(* IEC 61131-3 sources: Bob/Head_Pkg/ModuleControl, 4 files *)

(* ---- Types.typ ---- *)
TYPE
	PowerSupplyState_enum :
		(
		WAIT_FOR_READY_TO_POWER,
		WAIT_FOR_POWER_ON,
		READY,
		ERROR
		);
	localHead_typ : 	STRUCT
		pressureTransducerRaw : INT;
	END_STRUCT;
	localModule_typ : 	STRUCT
		ps : localPS_typ;
		valve : localValve_typ;
		supplyTemperatureRaw : INT;
		head : ARRAY[0..NUM_OF_HEADS_PER_MODULE_M1]OF localHead_typ;
	END_STRUCT;
	localPS_typ : 	STRUCT
		state : PowerSupplyState_enum;
		axis : ACP10AXIS_typ;
		mpAxis : UDINT;
		mpParams : MpAxisBasicParType;
		MpAxisBasic_0 : MpAxisBasic;
	END_STRUCT;
	localValve_typ : 	STRUCT
		valveName : STRING[80];
		outputModuleOk : BOOL; (*variable to be linked to the module ok on the IO module used for the outputs*)
		inputModuleOk : BOOL; (*variable to be linked to the module ok on the IO module used for the inputs*)
		doOpen : BOOL; (*variable to be linked to the digital output which opens the valve*)
		diOpened : BOOL; (*variable to be linked to the digital input which indicates that the valve is opened*)
		diClosed : BOOL; (*variable to be linked to the digital input which indicates that the valve is closed*)
		openDebounceTimer : TON;
		closeDebounceTimer : TON;
		openTime : REAL;
		openErrorTimer : TON;
		closeTime : REAL;
		closeErrorTimer : TON;
		MpRecipeRegPar_0 : MpRecipeRegPar;
		MpRecipeRegPar_1 : MpRecipeRegPar;
		openError_r_trig : r_trig;
		openError_f_trig : f_trig;
		closeError_r_trig : r_trig;
		closeError_f_trig : f_trig;
		open_and_close_error_r_trig : r_trig;
		open_and_close_error_f_trig : f_trig;
		io_error_r_trig : r_trig;
		io_error_f_trig : f_trig;
	END_STRUCT;
END_TYPE

(* ---- Main.st ---- *)
PROGRAM _INIT
    modules[0].valve.valveName := 'Module 1 Supply Valve';
    modules[1].valve.valveName := 'Module 2 Supply Valve';

    MpRecipeRegPar_0[0].PVName := ADR('gModules[0].heads[0].enable');
    MpRecipeRegPar_0[1].PVName := ADR('gModules[0].heads[1].enable');
    MpRecipeRegPar_0[2].PVName := ADR('gModules[1].heads[0].enable');
    MpRecipeRegPar_0[3].PVName := ADR('gModules[1].heads[1].enable');

    FOR currentHead:=0 TO NUMBER_OF_HEADS_M1 DO
        MpRecipeRegPar_0[currentHead].MpLink := ADR(gMachineRecipe);
        MpRecipeRegPar_0[currentHead].Enable := TRUE;
        MpRecipeRegPar_0[currentHead].Category := ADR(MACHINE_CATEGORY);
        MpRecipeRegPar_0[currentHead]();
    END_FOR

	gModules[0].productSupply.parameters;
    MpRecipeRegPar_1[0].PVName := ADR('gModules[0].productSupply.parameters');
    MpRecipeRegPar_1[1].PVName := ADR('gModules[1].productSupply.parameters');

    FOR currentHead:=0 TO NUMBER_OF_MODULES_M1 DO
        MpRecipeRegPar_1[currentHead].MpLink := ADR(gMachineRecipe);
        MpRecipeRegPar_1[currentHead].Enable := TRUE;
        MpRecipeRegPar_1[currentHead].Category := ADR(MACHINE_CATEGORY);
        MpRecipeRegPar_1[currentHead]();
    END_FOR

    MpRecipeRegPar_2[0].PVName := ADR('gModules[0].heads[0].pressureTransducer.parameters');
    MpRecipeRegPar_2[1].PVName := ADR('gModules[0].heads[1].pressureTransducer.parameters');
    MpRecipeRegPar_2[2].PVName := ADR('gModules[1].heads[0].pressureTransducer.parameters');
    MpRecipeRegPar_2[3].PVName := ADR('gModules[1].heads[1].pressureTransducer.parameters');

    FOR currentHead:=0 TO NUMBER_OF_HEADS_M1 DO
        MpRecipeRegPar_2[currentHead].MpLink := ADR(gMachineRecipe);
        MpRecipeRegPar_2[currentHead].Enable := TRUE;
        MpRecipeRegPar_2[currentHead].Category := ADR(MACHINE_CATEGORY);
        MpRecipeRegPar_2[currentHead]();
    END_FOR

END_PROGRAM

PROGRAM _CYCLIC

    memset(ADR(logArguments), 0, SIZEOF(logArguments));

	modules[0].ps.mpAxis := ADR(gMpAxisPS1);
	modules[1].ps.mpAxis := ADR(gMpAxisPS2);

	FOR currentModule:=0 TO NUMBER_OF_MODULES_M1 DO

        gModules[currentModule].productSupply.temperature   := ((modules[currentModule].supplyTemperatureRaw * gModules[currentModule].productSupply.parameters.scalingFactor) + gModules[currentModule].productSupply.parameters.scalingOffset) / 100.0;
        productSupplyValveAction;

        FOR currentHead:=0 TO NUM_OF_HEADS_PER_MODULE_M1 DO
			pCurrentHead ACCESS ADR(gModules[currentModule].heads[currentHead]);

			//set .ready bit for each head
            pCurrentHead.ready                          := ((pCurrentHead.stretchRod.status.atHome = TRUE OR pCurrentHead.stretchRod.status.atRetractPos= TRUE) AND (pCurrentHead.nozzle.status.opened = TRUE) AND ((pCurrentHead.fillPiston.status.atReturnPos = TRUE) OR (pCurrentHead.enable = FALSE)));
            pCurrentHead.pressureTransducer.pressure    := (modules[currentModule].head[currentHead].pressureTransducerRaw - pCurrentHead.pressureTransducer.parameters.scalingOffset) * pCurrentHead.pressureTransducer.parameters.scalingFactor;
        END_FOR

        logArguments[0] := ADR(currentModule);
        logArguments[1] := ADR(modules[currentModule].ps.MpAxisBasic_0.Info.HardwareInfo.NodeID);

        // if an error occurs in any state then go to the error state
        CASE modules[currentModule].ps.state OF
            ERROR:

            ELSE
                IF (modules[currentModule].ps.MpAxisBasic_0.Error = TRUE) THEN
                    logArguments[3] := ADR(modules[currentModule].ps.MpAxisBasic_0.StatusID);
                    logError('Power Supply', 'Module %h, Node %h Error %d', ADR(logArguments));
                    modules[currentModule].ps.state := ERROR;
                ELSIF (gModules[currentModule].powerSupply.commands.errorAcknowledge = TRUE) THEN
                    gModules[currentModule].powerSupply.commands.errorAcknowledge := FALSE;
                END_IF
        END_CASE

        CASE (modules[currentModule].ps.state) OF
            WAIT_FOR_READY_TO_POWER:
                IF (modules[currentModule].ps.MpAxisBasic_0.Info.AxisInitialized <> TRUE) AND (modules[currentModule].ps.MpAxisBasic_0.Update = FALSE) THEN
                    modules[currentModule].ps.MpAxisBasic_0.Update := TRUE;
                ELSIF (modules[currentModule].ps.MpAxisBasic_0.UpdateDone = TRUE) THEN
                    modules[currentModule].ps.MpAxisBasic_0.Update := FALSE;
                END_IF

                IF (modules[currentModule].ps.MpAxisBasic_0.Info.ReadyToPowerOn = TRUE) AND (gMachineControl.commands.powerOn = TRUE) THEN
					logArguments[0] := ADR(modules[currentModule].ps.MpAxisBasic_0.Info.HardwareInfo.NodeID);
					logDebug('PSControl', 'Power Supply Axis Ready to power on, index = %d', ADR(logArguments));
                    modules[currentModule].ps.MpAxisBasic_0.Power   := TRUE;
                    modules[currentModule].ps.state                 := WAIT_FOR_POWER_ON;
                END_IF

			WAIT_FOR_POWER_ON:
                IF (modules[currentModule].ps.MpAxisBasic_0.PowerOn = TRUE) THEN
                    logArguments[0] := ADR(modules[currentModule].ps.MpAxisBasic_0.Info.HardwareInfo.NodeID);
                    logDebug('PSControl', 'Node %d Power Supply Axis powered on', ADR(logArguments));
                    modules[currentModule].ps.state := READY;
                END_IF

            READY:
                IF (gMachineControl.commands.powerOn = FALSE) THEN
                    modules[currentModule].ps.MpAxisBasic_0.Power   := FALSE;
                    logArguments[0] := ADR(modules[currentModule].ps.MpAxisBasic_0.Info.HardwareInfo.NodeID);
                    logDebug('PSControl', 'Node %d Power Supply Axis powered off', ADR(logArguments));
                    modules[currentModule].ps.state := WAIT_FOR_READY_TO_POWER;
                END_IF

            ERROR:
                IF (gModules[currentModule].powerSupply.commands.errorAcknowledge = TRUE) THEN
                    logDebug('FillPiston', 'Module %h, Head %h, Node %h Acknowledging Error', ADR(logArguments));
                    gModules[currentModule].powerSupply.commands.errorAcknowledge   := FALSE;
                    modules[currentModule].ps.MpAxisBasic_0.ErrorReset                 := TRUE;
                END_IF

                IF (modules[currentModule].ps.MpAxisBasic_0.Error <> TRUE) THEN
                    logDebug('PSControl', 'Module %h, Node %h All Errors Acknowledged', ADR(logArguments));
                    modules[currentModule].ps.MpAxisBasic_0.ErrorReset  := FALSE;
                    IF (modules[currentModule].ps.MpAxisBasic_0.PowerOn = TRUE) THEN
                        modules[currentModule].ps.state := READY;
                    ELSE
                        modules[currentModule].ps.state := WAIT_FOR_READY_TO_POWER;
                    END_IF
                END_IF
        END_CASE

        IF (modules[currentModule].ps.state <> old_state[currentModule]) THEN
            old_state[currentModule] := modules[currentModule].ps.state;
            logArguments[0] := ADR(modules[currentModule].ps.MpAxisBasic_0.Info.HardwareInfo.NodeID);
            logArguments[1] := ADR(modules[currentModule].ps.state);
            logDebug('PSControl', 'Node %d Changing State to %d', ADR(logArguments));
        END_IF

        modules[currentModule].ps.MpAxisBasic_0.Enable      := TRUE;
        modules[currentModule].ps.MpAxisBasic_0.Axis        := ADR(modules[currentModule].ps.axis);
        modules[currentModule].ps.MpAxisBasic_0.MpLink      := modules[currentModule].ps.mpAxis;
        modules[currentModule].ps.MpAxisBasic_0.Parameters  := ADR(modules[currentModule].ps.mpParams);
        modules[currentModule].ps.MpAxisBasic_0();

        gModules[currentModule].powerSupply.status.errorActive  := modules[currentModule].ps.MpAxisBasic_0.Error;
        gModules[currentModule].powerSupply.status.errorNumber  := modules[currentModule].ps.MpAxisBasic_0.StatusID;
        gModules[currentModule].powerSupply.status.poweredOn    := modules[currentModule].ps.MpAxisBasic_0.PowerOn;

	END_FOR

END_PROGRAM

PROGRAM _EXIT
    FOR currentModule:=0 TO NUMBER_OF_MODULES_M1 DO
        modules[currentModule].ps.MpAxisBasic_0.Enable  := FALSE;
        modules[currentModule].ps.MpAxisBasic_0();
    END_FOR
END_PROGRAM

(* ---- productSupplyVavle.st ---- *)
ACTION productSupplyValveAction:

    pCurrentValve ACCESS ADR(gModules[currentModule].productSupply.valve);
    pLocalValve ACCESS ADR(modules[currentModule].valve);

    IF (pCurrentValve.parameters.machineData.enabled = TRUE) THEN

        IF (((pCurrentValve.commands.open = TRUE) AND (pCurrentValve.commands.close = FALSE)) AND
            (pLocalValve.doOpen = FALSE)) THEN
            logDebug('Fill Valve', 'Module %h, Head %h, Open Command', ADR(logArguments));
            pLocalValve.doOpen := TRUE;
        END_IF

        IF (((pCurrentValve.commands.close = TRUE) AND (pCurrentValve.commands.open = FALSE)) AND
            (pLocalValve.doOpen = TRUE)) THEN
            logDebug('Fill Valve', 'Module %h, Head %h, Close Command', ADR(logArguments));
            pLocalValve.doOpen := FALSE;
        END_IF

        // 20ms debounce timer
        pLocalValve.openDebounceTimer.IN    := pLocalValve.diOpened;
        pLocalValve.openDebounceTimer.PT    := pCurrentValve.parameters.machineData.debounceTime;
        pLocalValve.openDebounceTimer();

        // 20ms debounce timer
        pLocalValve.closeDebounceTimer.IN := pLocalValve.diClosed;
        pLocalValve.closeDebounceTimer.PT := pCurrentValve.parameters.machineData.debounceTime;
        pLocalValve.closeDebounceTimer();

        // ensure that the valve opens
        pLocalValve.openErrorTimer.IN    := ((pCurrentValve.commands.open = TRUE) AND (pLocalValve.diOpened = FALSE));
        pLocalValve.openErrorTimer.PT    := pCurrentValve.parameters.machineData.timeout;
        pLocalValve.openErrorTimer();

        // ensure that the valve closes
        pLocalValve.closeErrorTimer.IN := ((pCurrentValve.commands.close = TRUE) AND (pLocalValve.diClosed = FALSE));
        pLocalValve.closeErrorTimer.PT := pCurrentValve.parameters.machineData.timeout;
        pLocalValve.closeErrorTimer();

        pCurrentValve.status.opened             := pLocalValve.openDebounceTimer.Q;
        pCurrentValve.status.closed             := pLocalValve.closeDebounceTimer.Q;
        pCurrentValve.status.centered           := ((pCurrentValve.status.opened <> TRUE) AND (pCurrentValve.status.closed <> TRUE));
        pCurrentValve.status.position           := 0;
        pCurrentValve.status.fullFlowAchieved   := FALSE;

        pLocalValve.openError_r_trig.CLK := pLocalValve.openErrorTimer.Q;
        pLocalValve.openError_r_trig();
        IF (pLocalValve.openError_r_trig.Q = TRUE) THEN
            valveErrorName := pLocalValve.valveName;
            MpAlarmXSet(gAlarmXCore, 'VALVE_NOT_OPENED');
        END_IF
        pLocalValve.openError_f_trig.CLK := pLocalValve.openErrorTimer.Q;
        pLocalValve.openError_f_trig();
        IF (pLocalValve.openError_f_trig.Q = TRUE) THEN
            MpAlarmXReset(gAlarmXCore, 'VALVE_NOT_OPENED');
        END_IF

        pLocalValve.closeError_r_trig.CLK := pLocalValve.closeErrorTimer.Q;
        pLocalValve.closeError_r_trig();
        IF (pLocalValve.closeError_r_trig.Q = TRUE) THEN
            valveErrorName := pLocalValve.valveName;
            MpAlarmXSet(gAlarmXCore, 'VALVE_NOT_CLOSED');
        END_IF
        pLocalValve.closeError_f_trig.CLK := pLocalValve.closeErrorTimer.Q;
        pLocalValve.closeError_f_trig();
        IF (pLocalValve.closeError_f_trig.Q = TRUE) THEN
            MpAlarmXReset(gAlarmXCore, 'VALVE_NOT_CLOSED');
        END_IF

        pLocalValve.open_and_close_error_r_trig.CLK := ((pCurrentValve.commands.open = TRUE) AND (pCurrentValve.commands.close = TRUE));
        pLocalValve.open_and_close_error_r_trig();
        IF (pLocalValve.open_and_close_error_r_trig.Q = TRUE) THEN
            valveErrorName := pLocalValve.valveName;
            MpAlarmXSet(gAlarmXCore, 'VALVE_COMMANDED_OPEN_AND_CLOSE');
        END_IF
        pLocalValve.open_and_close_error_f_trig.CLK := ((pCurrentValve.commands.open = TRUE) AND (pCurrentValve.commands.close = TRUE));
        pLocalValve.open_and_close_error_f_trig();
        IF (pLocalValve.open_and_close_error_f_trig.Q = TRUE) THEN
            MpAlarmXReset(gAlarmXCore, 'VALVE_COMMANDED_OPEN_AND_CLOSE');
        END_IF

        pLocalValve.io_error_r_trig.CLK := ((pLocalValve.inputModuleOk = FALSE) OR (pLocalValve.outputModuleOk = FALSE));
        pLocalValve.io_error_r_trig();
        IF (pLocalValve.io_error_r_trig.Q = TRUE) THEN
            valveErrorName := pLocalValve.valveName;
            MpAlarmXSet(gAlarmXCore, 'VALVE_IO_MISSING');
        END_IF
        pLocalValve.io_error_f_trig.CLK := ((pLocalValve.inputModuleOk = FALSE) OR (pLocalValve.outputModuleOk = FALSE));
        pLocalValve.openError_f_trig();
        IF (pLocalValve.openError_f_trig.Q = TRUE) THEN
            MpAlarmXReset(gAlarmXCore, 'VALVE_IO_MISSING');
        END_IF

        pCurrentValve.status.errorActive        := NOT((pLocalValve.inputModuleOk AND pLocalValve.outputModuleOk)) OR
                                                      ((pLocalValve.closeErrorTimer.Q = TRUE) OR (pLocalValve.openErrorTimer.Q = TRUE)) OR
                                                      ((pCurrentValve.commands.open = TRUE) AND (pCurrentValve.commands.close = TRUE));

        IF (pCurrentValve.commands.errorAcknowledge = TRUE) THEN
            pCurrentValve.commands.errorAcknowledge := FALSE;
        END_IF
    END_IF

END_ACTION

(* ---- Variables.var ---- *)
VAR
	MpRecipeRegPar_0 : ARRAY[0..NUMBER_OF_HEADS_M1] OF MpRecipeRegPar;
	MpRecipeRegPar_1 : ARRAY[0..NUMBER_OF_MODULES_M1] OF MpRecipeRegPar;
	MpRecipeRegPar_2 : ARRAY[0..NUMBER_OF_HEADS_M1] OF MpRecipeRegPar;
	valveErrorName : STRING[80];
	pCurrentValve : REFERENCE TO valve_typ;
	pLocalValve : REFERENCE TO localValve_typ;
	modules : ARRAY[0..NUMBER_OF_MODULES_M1] OF localModule_typ;
	currentModule : USINT;
	logArguments : ARRAY[0..8] OF UDINT;
	old_state : {REDUND_UNREPLICABLE} ARRAY[0..NUMBER_OF_MODULES_M1] OF PowerSupplyState_enum;
	currentHead : USINT;
	pCurrentHead : REFERENCE TO FormingHead_typ;
END_VAR
